(* CODESYS project DairyTech_Molasses.project
   Title: DairyTech_Molasses
   Version: 0.0.0.0

Project tree, tasks and I/O mapping:
  MyController : TM218LDA24DRN, Schneider Electric, order no. TM218LDA24DRN, version 4.0.1.26
      settings: Expansion Tasks.Expansion 1 Task Name = 'MAST'
    application Application
      task MAST (cyclic, interval 20 ms, priority 15, watchdog 100 ms x 1) calls POU
      function HiddenPOU [ST]
      global variables GVL
      program POU [FBD]
    Embedded Functions
      IO : IO, Schneider Electric, version 4.0.1.26
          input  iwIO_IW0 : WORD  // IW0
          output qwIO_QW0 : WORD  // QW0
      HSC : HSC, Schneider Electric, version 4.0.1.26
    Serial Line 1
      Modbus_Manager_1 : Modbus Manager, Schneider Electric, version 4.0.0.2
    Serial Line 2
      Modbus_Manager : Modbus Manager, Schneider Electric, version 4.0.0.2
    Module_1 : TM2AMI4HTN, Schneider Electric, order no. TM2AMI4HTN, version 4.0.1.26
        settings: IW0.Maximum = 4000; IW1.Maximum = 15000
        input  iFlowMeter : INT  // IW0
        input  iPelletFeederRPM : INT  // IW1
        input  iiModule_1_IW2 : INT  // IW2
        input  iiModule_1_IW3 : INT  // IW3
*)

// MyController/Application/GVL
VAR_GLOBAL
	molassesFlowAct AT %MD0 : REAL;
	pelletFeederRPMAct AT %MD1 : REAL;
	setMolassesFlow AT %MD2 : REAL;
	oilPumpRPMCalc AT %MD3 : REAL;
	
	
	autoSel AT %MX100.0 : BOOL;

	pidReset AT %MX100.1 : BOOL;
	oilRPMFinal: WORD;
END_VAR

VAR_GLOBAL RETAIN
	feedFlowPerRev AT %MD10 : REAL;
	setMolassesPC AT %MD11 : REAL;
	oilPumpRPMManual AT %MD12 : REAL;
	pidGain AT %MD13 :REAL;
	pidDerivative AT %MD14 : REAL;
	pidIntegral AT %MD15 : REAL;
	
END_VAR

// MyController/Application/POU
PROGRAM POU
VAR
	feedFlowInKg: REAL;
	PID_0: PID;
	out: REAL;
	LIN_TRAFO_0: LIN_TRAFO;
	ADDM_0: ADDM;
	WRITE_VAR_0: WRITE_VAR;
	vfdAddr: ADDRESS;
	R_TRIG0: R_TRIG;
	busy1: BOOL;
	testOn: BOOL;
	oilPumpRPMPID: REAL;
END_VAR

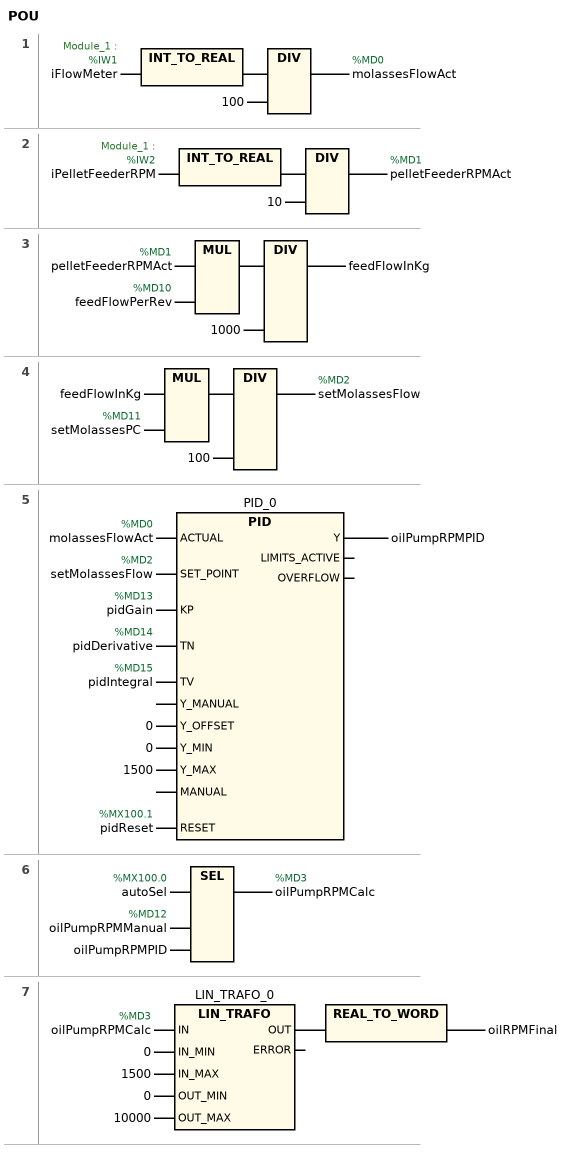
// NETWORK 1
//   iFlowMeter: Module_1 : | AT %IW1
//   molassesFlowAct: AT %MD0
molassesFlowAct := INT_TO_REAL(iFlowMeter) / 100;

// NETWORK 2
//   iPelletFeederRPM: Module_1 : | AT %IW2
//   pelletFeederRPMAct: AT %MD1
pelletFeederRPMAct := INT_TO_REAL(iPelletFeederRPM) / 10;

// NETWORK 3
//   pelletFeederRPMAct: AT %MD1
//   feedFlowPerRev: AT %MD10
feedFlowInKg := (pelletFeederRPMAct * feedFlowPerRev) / 1000;

// NETWORK 4
//   setMolassesPC: AT %MD11
//   setMolassesFlow: AT %MD2
setMolassesFlow := (feedFlowInKg * setMolassesPC) / 100;

// NETWORK 5
//   molassesFlowAct: AT %MD0
//   setMolassesFlow: AT %MD2
//   pidGain: AT %MD13
//   pidDerivative: AT %MD14
//   pidIntegral: AT %MD15
//   pidReset: AT %MX100.1
PID_0(
    ACTUAL := molassesFlowAct,
    SET_POINT := setMolassesFlow,
    KP := pidGain,
    TN := pidDerivative,
    TV := pidIntegral,
    Y_OFFSET := 0,
    Y_MIN := 0,
    Y_MAX := 1500,
    RESET := pidReset); // PID
oilPumpRPMPID := PID_0.Y;

// NETWORK 6
//   autoSel: AT %MX100.0
//   oilPumpRPMManual: AT %MD12
//   oilPumpRPMCalc: AT %MD3
oilPumpRPMCalc := SEL(autoSel, oilPumpRPMManual, oilPumpRPMPID);

// NETWORK 7
//   oilPumpRPMCalc: AT %MD3
LIN_TRAFO_0(IN := oilPumpRPMCalc, IN_MIN := 0, IN_MAX := 1500, OUT_MIN := 0, OUT_MAX := 10000); // LIN_TRAFO
oilRPMFinal := REAL_TO_WORD(LIN_TRAFO_0.OUT);

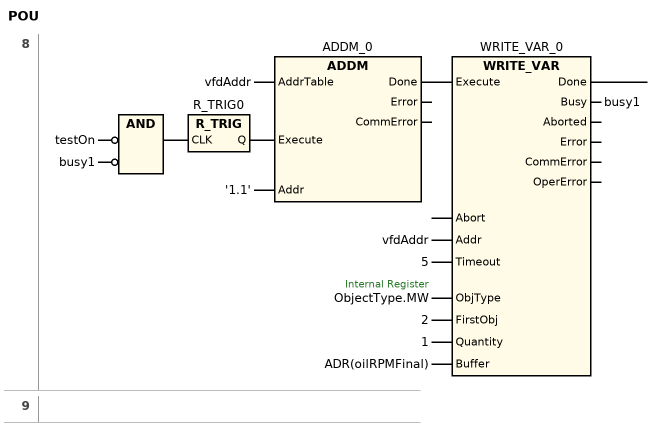
// NETWORK 8
//   ObjectType.MW: Internal Register
R_TRIG0(CLK := NOT testOn AND NOT busy1); // R_TRIG
ADDM_0(AddrTable := vfdAddr, Execute := R_TRIG0.Q, Addr := '1.1'); // ADDM
WRITE_VAR_0(
    Execute := ADDM_0.Done,
    Addr := vfdAddr,
    Timeout := 5,
    ObjType := ObjectType.MW,
    FirstObj := 2,
    Quantity := 1,
    Buffer := ADR(oilRPMFinal),
    Busy => busy1); // WRITE_VAR

// NETWORK 9

END_PROGRAM

// MyController/Application/HiddenPOU
FUNCTION HiddenPOU : BOOL

VAR_INPUT
	pHiddenFunc: POINTER TO WORD;
END_VAR
VAR
	pRead: POINTER TO BYTE;
	pWrite: POINTER TO BYTE;
END_VAR

pRead := pHiddenFunc + 400;
pWrite := pHiddenFunc + 4400;
HiddenPOU := TRUE;

END_FUNCTION
